{attribute 'OPC.UA.DA' := '1'}
FUNCTION_BLOCK PM101OpticalPowermeterHt EXTENDS PM101OpticalPowermeter
VAR_INPUT
END_VAR
VAR_OUTPUT
END_VAR
VAR
	{attribute 'OPC.UA.DA' := '0'}
	_config : PM101OpticalPowermeterConfig;
	{attribute 'OPC.UA.DA' := '0'}
	_polarisationConfig : PolarisationConfig;
	{attribute 'OPC.UA.DA' := '0'}
	_rFactorSettings : RFactorSettings;
	{attribute 'OPC.UA.DA' := '0'}
	_responsivityConfig : ResponsivityConfig;
	{attribute 'OPC.UA.DA' := '0'}
	_coeAccess : CoeAccess;
	{attribute 'OPC.UA.DA' := '0'}
	_initConfigSerialCom : BOOL;
	{attribute 'OPC.UA.DA' := '0'}	
	_serialCom  : SerialCom(Prefix :='', Suffix := Const.LINE_FEED);
	{attribute 'OPC.UA.DA' := '0'}
	_refSerialCom : REFERENCE TO SerialCom(Prefix :='', Suffix := Const.LINE_FEEL) := _serialCom;
	
	{attribute 'OPC.UA.DA' := '0'}
	_pulseGeneratorInit : TON;	
	{attribute 'OPC.UA.DA' := '0'}
	_itemInit : INT;
END_VAR

IF _config.IsSimulated THEN
	SUPER^(Conf := _config, PolarisationConfig := _polarisationConfig, RFactorSettings := _rfactorSettings, ResponsivityConfig := _responsivityConfig, SerialCom := _serialCom, RefSerialCom := _refSerialCom);
ELSE
	IF NOT InitConfigSerialCom THEN
		ConfigureSerialCom();
	ELSIF THIS^.Status = TExecutionState.Ready THEN
		IF _refSerialCom.ErrorReceiveId = COMERROR_NOERROR THEN
			_refSerialCom(TxBuffer:= HardwareGlobalVariables.TxBufferOpticalPowermeterHt, 
						  RxBuffer:= HardwareGlobalVariables.RxBufferOpticalPowermeterHt);
		END_IF	
					
		// Init device
		InitDevice(); 
  
		SUPER^(Conf := _config, PolarisationConfig := _polarisationConfig, RFactorSettings := _rfactorSettings, ResponsivityConfig := _responsivityConfig, SerialCom := _serialCom, RefSerialCom := _refSerialCom);							
	END_IF
END_IF

METHOD ConfigureSerialCom
VAR_INPUT
END_VAR
IF _coeAccess.CoeOperation.Ready THEN
	_logger.Information(_message.Reset().Append('Start configuration com serial').ToString());
END_IF;	

_coeAccess.CoeOperation.Start();
_coeAccess(SerialCommunication := _config.SerialCommunication);
	
IF _coeAccess.CoeOperation.Done THEN
	_coeAccess.SetDone();
	
	_Logger.Information(_message.Reset().
							Append('{').Append(TO_STRING(THIS^.Family)).Append('} : ').
							Append(' - Status : ').Append(TO_STRING(_coeAccess.Status)).ToString());
	InitConfigSerialCom := TRUE;
END_IF
 
IF _coeAccess.CoeOperation.Error THEN	
	_coeAccess.SetError(0);
	
	_Logger.Error(_message.Reset().
							Append('{').Append(TO_STRING(THIS^.Family)).Append('} : ').
							Append(' - Status : ').Append(TO_STRING(_coeAccess.Status)).ToString());
	InitConfigSerialCom := TRUE;
END_IF

THIS^.Status := _coeAccess.Status;
State := _coeAccess.Status;
END_METHOD

METHOD FB_init : BOOL
VAR_INPUT
	bInitRetains : BOOL; // if TRUE, the retain variables are initialized (warm start / cold start)
	bInCopyCode : BOOL;  // if TRUE, the instance afterwards gets moved into the copy code (online change)
	Config : PM101OpticalPowermeterConfig;
	PolarisationConfig : PolarisationConfig;
	RFactorSettings : RFactorSettings;
	ResponsivityConfig : ResponsivityConfig;
END_VAR
IF Config.IsEnabled THEN
	_config := Config;
	_polarisationConfig := PolarisationConfig;
	_rFactorSettings := RFactorSettings;
	_responsivityConfig := ResponsivityConfig;
	
	SUPER^._opticalPowermeterConfig.Name := Config.Name;
	SUPER^._opticalPowermeterConfig.DeviceID := Config.DeviceID;
	SUPER^._opticalPowermeterConfig.IsEnabled := Config.IsEnabled;
	SUPER^._opticalPowermeterConfig.LogLevel := Config.LogLevel;
	
	SUPER^.Name := Config.Name;
	SUPER^.DeviceID := Config.DeviceID;	
	THIS^.Family := DeviceFamily.OpticalPowermeter;
		
	_Logger.Information(_message.Reset().Append('Init ').
							Append('{').Append(TO_STRING(THIS^.Family)).Append('} - ').
							Append('{').Append(TO_STRING(Config.Name)).Append('}').ToString());																													
END_IF
END_METHOD

PROPERTY InitConfigSerialCom : BOOL
GET
InitConfigSerialCom := _initConfigSerialCom;
END_GET
SET
_initConfigSerialCom := InitConfigSerialCom;
END_SET
END_PROPERTY

METHOD InitDevice 
VAR_INPUT	
END_VAR
IF NOT _initDevice THEN	
	CASE _itemInit OF
		0:  _logger.Information(_message.Reset().Append(_config.Name).Append(' - InitDevice').ToString());
			_itemInit := 1;
		
		1:  SUPER^._rangeAuto := TRUE;
			SUPER^._cmdRange := 'TRUE';
			_itemInit := 2;			
			
		2:  SUPER^._setSensorAttenuation := TRUE;
			SUPER^._cmdSensorAttenuation := _config.Sensor.Attenuation;
			_itemInit := 3;
			
		3:  IF _config.Sensor.Name = Const.POWERMETER_SENSOR_NAME_S150C THEN
				_logger.Error(_message.Reset().Append(_config.Name).Append(' - Sensor name: ').Append(_config.Sensor.Name).ToString());
				_itemInit := 10;
			ELSIF _config.Sensor.Name = Const.POWERMETER_SENSOR_NAME_TAP_COUPLER THEN
				_logger.Error(_message.Reset().Append(_config.Name).Append(' - Sensor name: ').Append(_config.Sensor.Name).ToString());
				_itemInit := 20;
			ELSE
				_logger.Error(_message.Reset().Append(_config.Name).Append(' - NAME OF FAILED SENSOR').ToString());
		    END_IF
			
		10:  SUPER^._setWavelength := TRUE;
			 SUPER^._cmdWavelength := _config.Sensor.Wavelength;
			 _itemInit := 50;		
		
		20:  GetResponsivity();
			 _itemInit := 21;
			
		21:	 _pulseGeneratorInit(IN := TRUE, PT := T#3000MS);
			 IF _pulseGeneratorInit.Q THEN
				_pulseGeneratorInit(IN := FALSE);				
			 	_itemInit := 22;
			 END_IF
		
		22:	 IF ResponsivityMsg = LREAL_TO_STRING(_responsivityConfig.Responsivity_mA_W) THEN
			 	_logger.Information(_message.Reset().Append(_config.Name).Append(' - Responsivity already defined').ToString());
			 	_itemInit := 50;
			 ELSE				 
				_itemInit := 23;
			 END_IF	
			 
		23:  _logger.Information(_message.Reset().
							Append(_config.Name).
							Append(' - Init responsivity: ').
							Append(LREAL_TO_STRING(_responsivityConfig.Responsivity_mA_W)).ToString());
			
			SUPER^._setpoint := _responsivityConfig.Responsivity_ma_W;
			SUPER^._setResponsivity := TRUE;
			
			_itemInit := 50;

		50: _logger.Information(_message.Reset().
							Append(_config.Name).
							Append(' - InitDevice done').ToString());				
			_initDevice	:= TRUE;
	END_CASE			
END_IF
END_METHOD

END_FUNCTION_BLOCK

(* stored: Version 1.1.0.1, ProductVersion 3.1.4024.12
   POU PM101OpticalPowermeterHt: Id {e25f19f4-fdfc-4631-897f-437f7c79b736}, SpecialFunc None
   Folder Commands: Id {f350bd74-2873-4b2c-bf64-e2244013a150}
   Method ConfigureSerialCom: Id {7434936f-8635-46bc-b41e-38a9c328d528}
   Method FB_init: Id {e497c21b-666d-4718-9f85-5f33865cbb96}
   Property InitConfigSerialCom: Id {586176b1-6c27-45e2-bb12-0604a616e80d}
   Get Get: Id {9615dc4e-8676-4d13-856d-f0751a9d5c1f}
   Set Set: Id {4e319e66-1640-48f5-9fdf-48752e9f12e5}
   Method InitDevice: Id {11aebc39-96a6-4ae4-9757-4f031f341321} *)
